(* PLC project TEST.project, CODESYS CODESYS V3.5 SP3 Patch 7 *)
(* stored: creationDateTime 2013-12-19T09:52:46.2493553, modificationDateTime 2013-12-19T09:52:20.1898647 *)

FUNCTION_BLOCK Werkzeugtraeger
  VAR
    Motor : INT;
    Links : INT;
    Rechts : INT;
    Endlagenschalter : INT;
    Signal : INT;
  END_VAR

INITIAL_STEP WZT steht:
END_STEP
TRANSITION FROM WZT steht TO WZT dreht
  := Signal Motor;
END_TRANSITION
STEP WZT dreht:
END_STEP
TRANSITION FROM WZT dreht TO Init
  := Endlagenschalter 5;
END_TRANSITION
END_FUNCTION_BLOCK
